{attribute addProperty BoxType "EL6201-0000-0017"}
{attribute addProperty Id "Slave_17A_DO0BIT10.125129Slave_17A_DO1BIT10.125130Slave_17A_DO2BIT10.125131Slave_17A_DO3BIT10.125132Slave_17B_DO0BIT10.125133Slave_17B_DO1BIT10.125134Slave_17B_DO2BIT10.125135Slave_17B_DO3BIT10.125136"}
{attribute addProperty CRC "330413423"}
{attribute addProperty SizeInBites "8"}
{attribute addProperty SizeInBytes "1"}
TYPE Slave_17_Outputs_13B1B56F :
STRUCT
	{attribute addProperty Name "Slave_17A_DO0"}
	Slave_17A_DO0 : BIT;
	{attribute addProperty Name "Slave_17A_DO1"}
	Slave_17A_DO1 : BIT;
	{attribute addProperty Name "Slave_17A_DO2"}
	Slave_17A_DO2 : BIT;
	{attribute addProperty Name "Slave_17A_DO3"}
	Slave_17A_DO3 : BIT;
	{attribute addProperty Name "Slave_17B_DO0"}
	Slave_17B_DO0 : BIT;
	{attribute addProperty Name "Slave_17B_DO1"}
	Slave_17B_DO1 : BIT;
	{attribute addProperty Name "Slave_17B_DO2"}
	Slave_17B_DO2 : BIT;
	{attribute addProperty Name "Slave_17B_DO3"}
	Slave_17B_DO3 : BIT;
END_STRUCT
END_TYPE

(* stored: Version 1.2.0.0, ProductVersion 3.1.4024.9
   DUT Slave_17_Outputs_13B1B56F: Id {b0236504-de64-4559-9004-f3cca0abb758} *)
